(* CoDeSys 2.3 library: WAGOLibKNXDevice.lib *)

(* Data type *)
TYPE enumDeviceStatus :(
	KNX_DEVICE_NOT_INIT				:= 0, (*Device noch nicht initialisiert*)
	KNX_DEVICE_OK 					:= 1, (* OK *)
	KNX_APP_NOT_RUNNING 			:= 2, (* KNX Applikation laeuft nicht *)
	KNX_APPLICATION_LOADED 			:= 3, (* KNX Applikation wurde geladen *)
	KNX_APPLICATION_START_LOADING 	:= 4, (* KNX Applikation soll geladen werden *)
    KNX_APPL_CRC_OK 				:= 5, (* Checksumme ist OK *)
	KNX_APPL_CRC_ERR 				:= 6, (* Checksumme ist nicht OK *)
	KNX_APPL_SYS_ERR 				:= 7, (* KNX Applicationsfehler im Device *)
	KNX_DEVICE_KBUS_ERROR 			:= 8, (* KBus Fehler erkannt *)
	KNX_DEVICE_ETHERNET_ERROR 		:= 9);(* Ethernet Fehler erkannt, auf beiden Ports kein LINK *)
END_TYPE

(* Data type *)
TYPE typDeviceStatus :
STRUCT
	eDeviceStatus : enumDeviceStatus;
	bDeviceProgMode: BYTE;
END_STRUCT
END_TYPE

(* POU GET_DEVICE_STATUS, ST *)
FUNCTION_BLOCK GET_DEVICE_STATUS
(*******************************************************************************
   WAGO Kontakttechnik GmbH & Co. KG Hansastr. 27 32423 Minden(Westf.) 
  Tel. +49571/887-0              
                                                                                  
  Function: GET_DEVICE_STATUS
 
  Version:	1.0
  Date: 		23.01.2008
*******************************************************************************)

VAR_INPUT
END_VAR
VAR_OUTPUT
	stDeviceStatue : typDeviceStatus;
END_VAR
VAR
END_VAR
;
END_FUNCTION_BLOCK

(* POU KNXDeviceCRC, ST *)
FUNCTION KNXDeviceCRC: BOOL
(*******************************************************************************
   WAGO Kontakttechnik GmbH & Co. KG Hansastr. 27 32423 Minden(Westf.) 
  Tel. +49571/887-0              
                                                                                  
  Function: KNXDeviceCRC
 
  Version:	1.0
  Date: 		23.01.2008
*******************************************************************************)
VAR_INPUT
	dwCRC: DWORD;
END_VAR
;
END_FUNCTION
